Universal Robots PolyScope program: 20250526log.urp

Program 20250526log (installation=20240827 directory=/programs/collection createdIn=5.15.1 lastSavedIn=5.15.1 robotSerialNumber=20245500285)
Calibrated DH parameters: a=[0.000097, -0.210459, -0.026602, 0.000137, 0.000078, 0]; d=[0.162601, 254.180657, -54.076236, -199.970743, 0.099615, 0.099684]; alpha=[1.569796, -0.001455, 0.001957, 1.570525, -1.571561, 0]; deltaTheta=[0, -1.053331, 8.839472, -1.50296, 0.000002, 0]
InitVariablesNode
Robot Program (runOnlyOnce=false)
  Popup Message (haltProgram=false message=gf225_multi_recon3d-20250526log.py inputType=Text)
  '0-空闲/1-接触面验证/2-中心点Z/22-无人看守中心点Z/3-全点Z/33-无人看守全点Z'
  mode := 22
  step_x := 0.004
  step_y := 0.004
  step_z := 0.0002
  step_tcp := 0.0001
  '二维数组xy(0,0)(-1,-1)(1,1)(-1,1)(1,-1)(0,0)'
  var_x := [0,-1,1,-1,1,0]
  var_y := [0,-1,1,1,-1,0]
  '设置端口 192.168.1.7:9125'
  Script: pc_code = rpc_factory("xmlrpc","http://192.168.1.7:9125/RPC2")
  MoveJ speed 60 deg/s, acceleration 80 deg/s^2 (useActiveTCP=true) feature=Base
    Waypoint 安全点: TCP in base x=97.16 y=948.75 z=68.916 mm, rx=0.003 ry=-2.2174 rz=-2.2186 rad; joints [249.762, -15.837, 68.005, -232.195, -69.643, 179.994] deg; TCP offset x=-0.17 y=0 z=192.95 mm, rx=0 ry=0 rz=0 rad
    SuppressedNode
      Waypoint 路点_1: 
    Waypoint 接触点: TCP in base x=97.126 y=948.749 z=64.69 mm, rx=0.003 ry=-2.2174 rz=-2.2186 rad; joints [249.763, -15.353, 67.701, -232.374, -69.641, 179.993] deg
    SuppressedNode
      Waypoint 路点_2: 
  If mode==0
    Popup Warning (haltProgram=false message=选择模式mode值 inputType=Text)
  ElseIf mode==1
    Popup Message (haltProgram=false message=1-接触面验证 inputType=Text)
    step := 0
    Loop Counting (count=30) loopVariable(name=循环_1)
      step := step+1
      tcp := pose_add(接触点, p[0,0,-step_tcp*step,0,0,0])
      tcpx := tcp[0]
      tcpy := tcp[1]
      tcpz := tcp[2]
      Popup Message (haltProgram=false inputType=Variable) variable=tcp
      MoveJ speed 60 deg/s, acceleration 80 deg/s^2 (useActiveTCP=true) feature=Base
        Waypoint Variable (Variable): variable=tcp
    Popup Message (haltProgram=false message=1-接触面验证完成 inputType=Text)
  ElseIf mode==2
    Popup Message (haltProgram=false message=2-中心点Z测试 inputType=Text)
    step := 0
    Loop Counting (count=20) loopVariable(name=循环_2)
      step := step+1
      Popup Message (haltProgram=false inputType=Variable) variable=step
      tcp := pose_add(接触点, p[0,0,-step_z*step,0,0,0])
      tcpx := tcp[0]
      tcpy := tcp[1]
      tcpz := tcp[2]
      MoveJ speed 60 deg/s, acceleration 80 deg/s^2 (useActiveTCP=true) feature=Base
        Popup Message (haltProgram=false inputType=Variable) variable=tcpz
        Waypoint Variable (Variable): variable=tcp
      Script: pc_code.xyz_s(tcpx,tcpy,tcpz)
      Wait Sleep waitTime=7
    MoveJ speed 60 deg/s, acceleration 80 deg/s^2 (useActiveTCP=true) feature=Base
      Waypoint 安全点: TCP in base x=97.16 y=948.75 z=68.916 mm, rx=0.003 ry=-2.2174 rz=-2.2186 rad; joints [249.762, -15.837, 68.005, -232.195, -69.643, 179.994] deg
    Popup Message (haltProgram=false message=2-中心点Z测试完成 inputType=Text)
  ElseIf mode==22
    Popup Message (haltProgram=false message=22-中心点Z自动测试 inputType=Text)
    step := 0
    Loop Counting (count=20) loopVariable(name=循环_3)
      step := step+1
      SuppressedNode
        Popup Message (haltProgram=false inputType=Variable) variable=step
      tcp := pose_add(接触点, p[0,0,-step_z*step,0,0,0])
      tcpx := tcp[0]
      tcpy := tcp[1]
      tcpz := tcp[2]
      MoveJ speed 60 deg/s, acceleration 80 deg/s^2 (useActiveTCP=true) feature=Base
        SuppressedNode
          Popup Message (haltProgram=false inputType=Variable) variable=tcpz
        Waypoint Variable (Variable): variable=tcp
      Wait Sleep waitTime=1
      Script: pc_code.xyz_s(tcpx,tcpy,tcpz)
      Wait Sleep waitTime=9
    MoveJ speed 60 deg/s, acceleration 80 deg/s^2 (useActiveTCP=true) feature=Base
      Waypoint 安全点: TCP in base x=97.16 y=948.75 z=68.916 mm, rx=0.003 ry=-2.2174 rz=-2.2186 rad; joints [249.762, -15.837, 68.005, -232.195, -69.643, 179.994] deg
    Popup Message (haltProgram=false message=22-中心点Z自动测试完成 inputType=Text)
  ElseIf mode==3
    Popup Message (haltProgram=false message=3-全点Z测试 inputType=Text)
    var_xy := 0
    Loop Counting (count=5) loopVariable(name=循环_5)
      MoveJ speed 60 deg/s, acceleration 80 deg/s^2 (useActiveTCP=true) feature=Base
        Waypoint 安全点: TCP in base x=97.16 y=948.75 z=68.916 mm, rx=0.003 ry=-2.2174 rz=-2.2186 rad; joints [249.762, -15.837, 68.005, -232.195, -69.643, 179.994] deg
      var_xy := var_xy+1
      step := 0
      Loop Counting (count=20) loopVariable(name=循环_6)
        step := step+1
        Popup Message (haltProgram=false inputType=Variable) variable=step
        tcp := pose_add(接触点, p[step_x*var_x[var_xy],step_y*var_y[var_xy],-step_z*step,0,0,0])
        tcpx := tcp[0]
        tcpy := tcp[1]
        tcpz := tcp[2]
        MoveJ speed 60 deg/s, acceleration 80 deg/s^2 (useActiveTCP=true) feature=Base
          Popup Message (haltProgram=false inputType=Variable) variable=tcpz
          Waypoint Variable (Variable): variable=tcp
        Script: pc_code.xyz_s(tcpx,tcpy,tcpz)
        Wait Sleep waitTime=7
      Popup Message (haltProgram=false inputType=Variable) variable=tcp
    MoveJ speed 60 deg/s, acceleration 80 deg/s^2 (useActiveTCP=true) feature=Base
      Waypoint 安全点: TCP in base x=97.16 y=948.75 z=68.916 mm, rx=0.003 ry=-2.2174 rz=-2.2186 rad; joints [249.762, -15.837, 68.005, -232.195, -69.643, 179.994] deg
    Popup Message (haltProgram=false message=3-全点Z测试完成 inputType=Text)
  ElseIf mode==33
    Popup Message (haltProgram=false message=33-全点Z自动测试 inputType=Text)
    var_xy := 0
    Loop Counting (count=5) loopVariable(name=循环_4)
      MoveJ speed 60 deg/s, acceleration 80 deg/s^2 (useActiveTCP=true) feature=Base
        Waypoint 安全点: TCP in base x=97.16 y=948.75 z=68.916 mm, rx=0.003 ry=-2.2174 rz=-2.2186 rad; joints [249.762, -15.837, 68.005, -232.195, -69.643, 179.994] deg
      var_xy := var_xy+1
      step := 0
      Loop Counting (count=20) loopVariable(name=循环_7)
        step := step+1
        SuppressedNode
          Popup Message (haltProgram=false inputType=Variable) variable=step
        tcp := pose_add(接触点, p[step_x*var_x[var_xy],step_y*var_y[var_xy],-step_z*step,0,0,0])
        tcpx := tcp[0]
        tcpy := tcp[1]
        tcpz := tcp[2]
        MoveJ speed 60 deg/s, acceleration 80 deg/s^2 (useActiveTCP=true) feature=Base
          SuppressedNode
            Popup Message (haltProgram=false inputType=Variable) variable=tcpz
          Waypoint Variable (Variable): variable=tcp
        Wait Sleep waitTime=1
        Script: pc_code.xyz_s(tcpx,tcpy,tcpz)
        Wait Sleep waitTime=9
      SuppressedNode
        Popup Message (haltProgram=false inputType=Variable) variable=tcp
    MoveJ speed 60 deg/s, acceleration 80 deg/s^2 (useActiveTCP=true) feature=Base
      Waypoint 安全点: TCP in base x=97.16 y=948.75 z=68.916 mm, rx=0.003 ry=-2.2174 rz=-2.2186 rad; joints [249.762, -15.837, 68.005, -232.195, -69.643, 179.994] deg
    Popup Message (haltProgram=false message=33-全点Z自动测试完成 inputType=Text)
